INTERFACE I_DatatypePack

METHOD RegisterWith
VAR_INPUT
	Datatypes : I_Datatypes;
END_VAR
END_METHOD

END_INTERFACE

(* stored: Version 1.1.0.1, ProductVersion 3.1.4024.12
   Itf I_DatatypePack: Id {509b29d4-db31-0acc-1617-f43ec2a97095}
   Method RegisterWith: Id {a7f18cec-c752-01f8-2962-81a2935f88e1} *)
